TYPE RFID :
STRUCT
END_STRUCT
END_TYPE

(* stored: Version 1.1.0.1, ProductVersion 3.1.4024.12
   DUT RFID: Id {e317f65a-fd59-4351-9b20-d10ee4ec149b} *)
